# EPICS autosave request: CARSApp/Db/DAC_AMVE-9210_settings.req
# Copy of VME_DAC_settings.req to go along with DAC.db
$(P)$(DAC)_1.DESC
$(P)$(DAC)_1.DRVH
$(P)$(DAC)_1.DRVL
$(P)$(DAC)_1_tweakVal.VAL
$(P)$(DAC)_2.DESC
$(P)$(DAC)_2.DRVH
$(P)$(DAC)_2.DRVL
$(P)$(DAC)_2_tweakVal.VAL
$(P)$(DAC)_3.DESC
$(P)$(DAC)_3.DRVH
$(P)$(DAC)_3.DRVL
$(P)$(DAC)_3_tweakVal.VAL
$(P)$(DAC)_4.DESC
$(P)$(DAC)_4.DRVH
$(P)$(DAC)_4.DRVL
$(P)$(DAC)_4_tweakVal.VAL
$(P)$(DAC)_5.DESC
$(P)$(DAC)_5.DRVH
$(P)$(DAC)_5.DRVL
$(P)$(DAC)_5_tweakVal.VAL
$(P)$(DAC)_6.DESC
$(P)$(DAC)_6.DRVH
$(P)$(DAC)_6.DRVL
$(P)$(DAC)_6_tweakVal.VAL
$(P)$(DAC)_7.DESC
$(P)$(DAC)_7.DRVH
$(P)$(DAC)_7.DRVL
$(P)$(DAC)_7_tweakVal.VAL
$(P)$(DAC)_8.DESC
$(P)$(DAC)_8.DRVH
$(P)$(DAC)_8.DRVL
$(P)$(DAC)_8_tweakVal.VAL

$(P)$(DAC)_1.VAL
$(P)$(DAC)_2.VAL
$(P)$(DAC)_3.VAL
$(P)$(DAC)_4.VAL
$(P)$(DAC)_5.VAL
$(P)$(DAC)_6.VAL
$(P)$(DAC)_7.VAL
$(P)$(DAC)_8.VAL
